Omron CX-Programmer project NewProject (CX-Programmer 9.70)

# PLC NewPLC1: CP1E E20

## Global symbols (name address type ; comment)
0.00 BOOL  ; START\STOP
0.01 BOOL  ; START/STOP
0.05 BOOL  ; START/STOP
100.00 BOOL  ; LED

## Program NewProgram1 (cyclic task 0)

### Section Section1

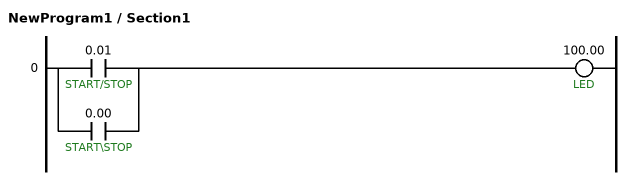
; rung 0
LD 0.01  ; START/STOP
OR 0.00  ; START\STOP
OUT 100.00  ; LED

### Section END
; rung 0
END(001)